// TIA Portal V18 export
// export: Created 2026-04-18T00:00:00Z, ExportSetting WithDefaults
ORGANIZATION_BLOCK "Main"   // OB1, LAD, ProgramCycle
{ S7_Optimized_Access := 'TRUE' }
VERSION : 0.1
// stored: AutoNumber true, IsIECCheckEnabled false
   VAR_INPUT
      Initial_Call : Bool;
      Remanence : Bool;
   END_VAR
BEGIN

REGION Network 1: Gọi khối mô phỏng cảm biến SCADA
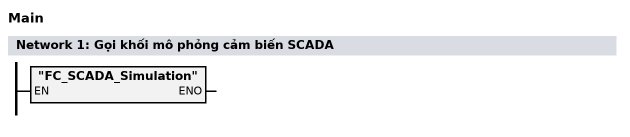
   RUNG wire#powerrail
      "FC_SCADA_Simulation"()
   END_RUNG
   // the same network as SCL:
   "FC_SCADA_Simulation"();
END_REGION
END_ORGANIZATION_BLOCK
